// TIA Portal V18 export
TYPE "Changeover_ShW"
// stored: IsFailsafeCompliant false
   STRUCT
      AutoDownloadTrigger : Bool;
      ManualDownloadTrigger : Bool;
      Result : Int;
      Completed : Bool;
   END_STRUCT;
END_TYPE
